// TIA Portal project "BarcodeScanner" (V12)

(* hardware
DEVICE "S7-1200 station_1"  SIMATIC 1200-Station
   slot 0: "S7-1200 rack"  Rack  V1.0
   slot 1: "PLC_1"  CPU 1212C DC/DC/Rly  6ES7 212-1HD30-0XB0  V2.2
*)

// ===== PLC "PLC_1"  CPU 1212C DC/DC/Rly =====

VAR_GLOBAL   // PLC tag table "Default tag table"
   "DI02" AT %I0.1 : Bool;
   "DI01" AT %I0.0 : Bool;
   "AI01" AT %IW64 : Int;
   "DO01" AT %Q0.0 : Bool;
   "DO02" AT %Q0.1 : Bool;
   "Counter1" AT %MW0 : Int;
   "Counter2" AT %MW2 : Int;
   "AI01Scaled" AT %MD10 : Real;
   "CounterAI" AT %M12.0 : Bool;
END_VAR

DATA_BLOCK "DB1"   // DB1
{ S7_Optimized_Access := 'FALSE' }
VERSION : 0.1
   VAR
      Machine1Motor : Bool;
      Machine2Motor : Bool;
      Machine1CounterSensor : Bool;
      Machine2CounterSensor : Bool;
      Machine1Counter : Int := 0;
      Machine2Counter : Int;
      Machine1ResetCounter : Bool;
      Machine2ResetCounter : Bool;
      Machine1CounterAI : Int;
      Barcode1Counter : Int;
      Barcode2Counter : Int;
      Machine1Counter_2 : Int;
      Machine2Counter_2 : Int;
   END_VAR
BEGIN
END_DATA_BLOCK

// folder: System blocks/Program resources

DATA_BLOCK "Machine01Counter1"   // DB2
{ S7_Optimized_Access := 'FALSE' }
AUTHOR : Simatic
FAMILY : IEC
NAME : CNTR
VERSION : 1.0
// stored: InstanceOfName ?
"?"
BEGIN
END_DATA_BLOCK

DATA_BLOCK "Machine02Counter2"   // DB3
{ S7_Optimized_Access := 'FALSE' }
AUTHOR : Simatic
FAMILY : IEC
NAME : CNTR
VERSION : 1.0
// stored: InstanceOfName ?
"?"
BEGIN
END_DATA_BLOCK

DATA_BLOCK "CounterMachine1AI"   // DB4
{ S7_Optimized_Access := 'FALSE' }
AUTHOR : Simatic
FAMILY : IEC
NAME : CNTR
VERSION : 1.0
// stored: InstanceOfName ?
"?"
BEGIN
END_DATA_BLOCK

// folder: (top level)

FUNCTION "StopMachine2WhenBlank" : Void   // FC1, SCL
{ S7_Optimized_Access := 'FALSE' }
VERSION : 0.1
BEGIN
   IF ABS("DB1".Barcode2Counter-"DB1".Machine2Counter)>1 THEN
     "DB1".Machine2Motor:=true;
     "DB1".Barcode2Counter := "DB1".Machine2Counter;
   END_IF;
END_FUNCTION

FUNCTION "StopMachine1WhenBlank" : Void   // FC2, SCL
{ S7_Optimized_Access := 'FALSE' }
VERSION : 0.1
BEGIN
   IF ABS("DB1".Barcode1Counter-"DB1".Machine1Counter)>1 THEN
     "DB1".Machine1Motor:=true;
     "DB1".Barcode1Counter := "DB1".Machine1Counter;
   END_IF;
END_FUNCTION

ORGANIZATION_BLOCK "Main"   // OB1, LAD, ProgramCycle
TITLE = "Main Program Sweep (Cycle)"
{ S7_Optimized_Access := 'FALSE' }
VERSION : 0.1
BEGIN

REGION Network 1
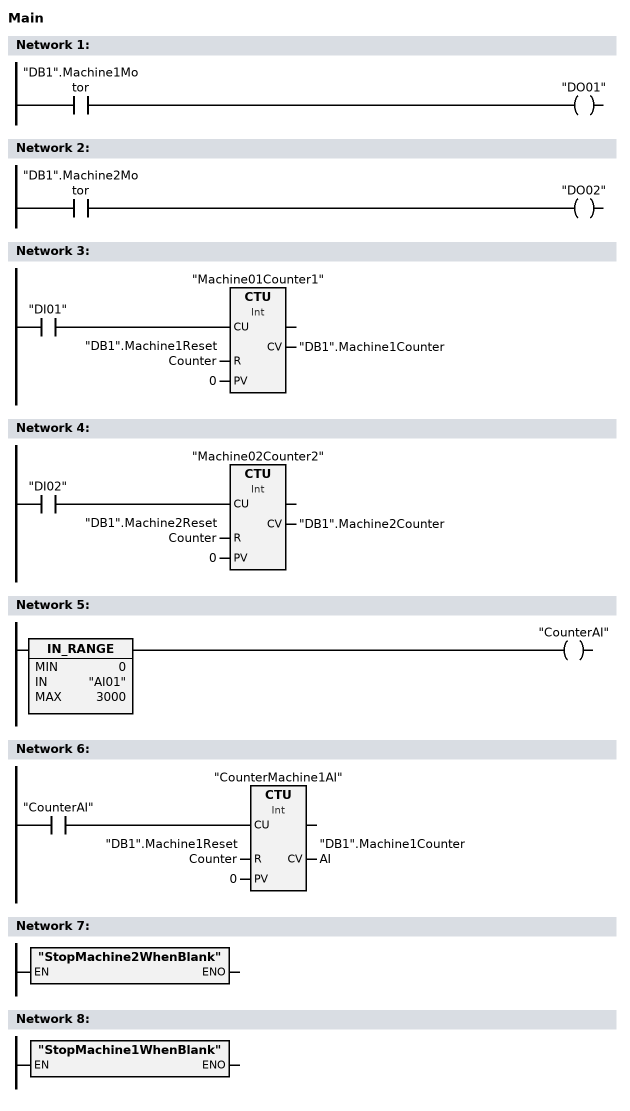
   RUNG wire#powerrail
      Contact( "DB1".Machine1Motor )
      Coil( "DO01" )
   END_RUNG
   // the same network as SCL:
   "DO01" := "DB1".Machine1Motor;
END_REGION

REGION Network 2
   RUNG wire#powerrail
      Contact( "DB1".Machine2Motor )
      Coil( "DO02" )
   END_RUNG
   // the same network as SCL:
   "DO02" := "DB1".Machine2Motor;
END_REGION

REGION Network 3
   "Machine01Counter1".CTU(CU := "DI01", R := "DB1".Machine1ResetCounter, PV := 0, CV => "DB1".Machine1Counter);
END_REGION

REGION Network 4
   "Machine02Counter2".CTU(CU := "DI02", R := "DB1".Machine2ResetCounter, PV := 0, CV => "DB1".Machine2Counter);
END_REGION

REGION Network 5
   RUNG wire#powerrail
      { S7_Templates := "SrcType := Int" } InRange(min := 0, in := "AI01", max := 3000)
      Coil( "CounterAI" )
   END_RUNG
   // the same network as SCL:
   "CounterAI" := (0 <= "AI01") AND ("AI01" <= 3000);
END_REGION

REGION Network 6
   "CounterMachine1AI".CTU(CU := "CounterAI",
                           R := "DB1".Machine1ResetCounter,
                           PV := 0,
                           CV => "DB1".Machine1CounterAI);
END_REGION

REGION Network 7
   RUNG wire#powerrail
      "StopMachine2WhenBlank"()
   END_RUNG
   // the same network as SCL:
   "StopMachine2WhenBlank"();
END_REGION

REGION Network 8
   RUNG wire#powerrail
      "StopMachine1WhenBlank"()
   END_RUNG
   // the same network as SCL:
   "StopMachine1WhenBlank"();
END_REGION
END_ORGANIZATION_BLOCK